SUBAPPLICATION InnerSubApp (* Subapplication Type *)
  (* Standard: 61499-2 *)
  (* Version 1.0, 2024-08-05, mario *)
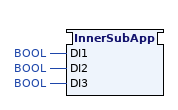
  VAR_INPUT
    DI1 : BOOL := FALSE;
    DI2 : BOOL := TRUE;
    DI3 : BOOL := TRUE;
  END_VAR
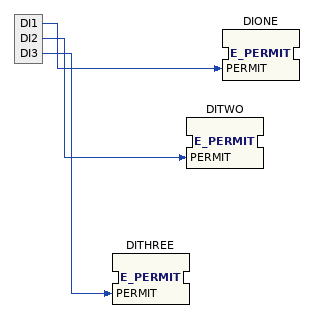
  FBS
    DIONE : E_PERMIT;
    DITWO : E_PERMIT;
    DITHREE : E_PERMIT;
  END_FBS
  DATA_CONNECTIONS
    DI1 TO DIONE.PERMIT;
    DI2 TO DITWO.PERMIT;
    DI3 TO DITHREE.PERMIT;
  END_CONNECTIONS
END_SUBAPPLICATION
